// TIA Portal V20 export
VAR_GLOBAL   // PLC tag table "Servo Telgram"
   BA010AZCRDR1_UnwinderLeftAxisT_Actor_Interface_AddressIn AT %I5114.0 : "PD_TEL105_IN";
   BA010AZCRDR1_UnwinderLeftAxisT_Actor_Interface_TorqueDataAddressIn AT %I5134.0 : "PD_TEL750_IN";
   BA010AZCRDR2_UnwinderRightAxisT_Actor_Interface_AddressIn AT %I5214.0 : "PD_TEL105_IN";
   BA010AZCRDR2_UnwinderRightAxisT_Actor_Interface_TorqueDataAddressIn AT %I5234.0 : "PD_TEL750_IN";
   BA010AZCRDR3_CompensatorAxisZ_Actor_Interface_AddressIn AT %I5314.0 : "PD_TEL105_IN";
   BA010AZCRDR3_CompensatorAxisZ_Actor_Interface_TorqueDataAddressIn AT %I5344.0 : "PD_TEL750_IN";
   BA010AZCRDR4_FeedingRollAxisT_Actor_Interface_AddressIn AT %I5414.0 : "PD_TEL105_IN";
   BA010AZCRDR5_ElectordCutterAxisZ_Actor_Interface_AddressIn AT %I5514.0 : "PD_TEL105_IN";
   BA010AZCRDR6_PositionMovingAxisX_Actor_Interface_AddressIn AT %I5614.0 : "PD_TEL105_IN";
   "BA010AZCRDR7_NG&ManualInputAxisY_Actor_Interface_AddressIn" AT %I5714.0 : "PD_TEL105_IN";
   BA010AZCRDR8_MagazineAxisZ_Actor_Interface_AddressIn AT %I5814.0 : "PD_TEL105_IN";
   BA010AZCRDR9_VisionAxisZ_Actor_Interface_AddressIn AT %I5914.0 : "PD_TEL105_IN";
   BA010AZCRDR16_ReelcutRingBlow_Actor_Interface_AddressIn AT %I9906.0 : "LPD_typePDTel352In";
   BA010AZCRDR17_StackRingBlow_Actor_Interface_AddressIn AT %I9924.0 : "LPD_typePDTel352In";
   BA010AZCRDR18_StackRingBlow_Actor_Interface_AddressIn AT %I9942.0 : "LPD_typePDTel352In";
   BA010AZCRDR2_UnwinderRightAxisT_Actor_Interface_TorqueDataAddressOut AT %Q5234.0 : "PD_TEL750_OUT";
   BA010AZCRDR3_CompensatorAxisZ_Actor_Interface_TorqueDataAddressOut AT %Q5344.0 : "PD_TEL750_OUT";
   BA010AZCRDR1_UnwinderLeftAxisT_Actor_Interface_TorqueDataAddressOut AT %Q5134.0 : "PD_TEL750_OUT";
   BA010AZCRDR1_UnwinderLeftAxisT_Actor_Interface_AddressOut AT %Q5114.0 : "PD_TEL105_OUT";
   BA010AZCRDR9_VisionAxisZ_Actor_Interface_AddressOut AT %Q5914.0 : "PD_TEL105_OUT";
   BA010AZCRDR2_UnwinderRightAxisT_Actor_Interface_TAddressOut AT %Q5214.0 : "PD_TEL105_OUT";
   BA010AZCRDR8_MagazineAxisZ_Actor_Interface_AddressOut AT %Q5814.0 : "PD_TEL105_OUT";
   BA010AZCRDR3_CompensatorAxisZ_Actor_Interface_AddressOut AT %Q5314.0 : "PD_TEL105_OUT";
   BA010AZCRDR4_FeedingRollAxisT_Actor_Interface_AddressOut AT %Q5414.0 : "PD_TEL105_OUT";
   "BA010AZCRDR7_NG&ManualInputAxisY_Actor_Interface_AddressOut" AT %Q5714.0 : "PD_TEL105_OUT";
   BA010AZCRDR5_ElectordCutterAxisZ_Actor_Interface_AddressOut AT %Q5514.0 : "PD_TEL105_OUT";
   BA010AZCRDR6_PositionMovingAxisX_Actor_Interface_AddressOut AT %Q5614.0 : "PD_TEL105_OUT";
   BA010AZCRDR17_StackRingBlow_Actor_Interface_AddressOut AT %Q9924.0 : "LPD_typePDTel352Out";
   BA010AZCRDR18_StackRingBlow_Actor_Interface_AddressOut AT %Q9942.0 : "LPD_typePDTel352Out";
   BA010AZCRDR16_ReelcutRingBlow_Actor_Interface_AddressOut AT %Q9906.0 : "LPD_typePDTel352Out";
   BA010AZCRDR10_NgKickerAxisZ_Actor_Interface_AddressIn AT %I6014.0 : "PD_TEL105_IN";
   BA010AZCRDR10_NgKickerAxisZ_Actor_Interface_AddressOut AT %Q6014.0 : "PD_TEL105_OUT";
   BA010AZCRDR10_NgKickerAxisZ_Actor_Interface_TorqueDataAddressIn AT %I476.0 : "PD_TEL750_IN";
   BA010AZCRDR10_NgKickerAxisZ_Actor_Interface_TorqueDataAddressOut AT %Q476.0 : "PD_TEL750_OUT";
   BA010AZCRDR11_PassKickerAxisZ_Actor_Interface_AddressIn AT %I6114.0 : "PD_TEL105_IN";
   BA010AZCRDR11_PassKickerAxisZ_Actor_Interface_AddressOut AT %Q6114.0 : "PD_TEL105_OUT";
   BA010AZCRDR11_PassKickerAxisZ_Actor_Interface_TorqueDataAddressIn AT %I702.0 : "PD_TEL750_IN";
   BA010AZCRDR11_PassKickerAxisZ_Actor_Interface_TorqueDataAddressOut AT %Q702.0 : "PD_TEL750_OUT";
   BA010AZCRDR12_CutConveyorAxisB_Actor_Interface_AddressIn AT %I6214.0 : "PD_TEL105_IN";
   BA010AZCRDR12_CutConveyorAxisB_Actor_Interface_AddressOut AT %Q6214.0 : "PD_TEL105_OUT";
   BA010AZCRDR12_CutConveyorAxisB_Actor_Interface_TorqueDataAddressIn AT %I6234.0 : "PD_TEL750_IN";
   BA010AZCRDR12_CutConveyorAxisB_Actor_Interface_TorqueDataAddressOut AT %Q6234.0 : "PD_TEL750_OUT";
   BA010AZCRDR13_NgConveyorAxisB_Actor_Interface_AddressIn AT %I6314.0 : "PD_TEL105_IN";
   BA010AZCRDR13_NgConveyorAxisB_Actor_Interface_AddressOut AT %Q6314.0 : "PD_TEL105_OUT";
   BA010AZCRDR13_NgConveyorAxisB_Actor_Interface_TorqueDataAddressIn AT %I6334.0 : "PD_TEL750_IN";
   BA010AZCRDR13_NgConveyorAxisB_Actor_Interface_TorqueDataAddressOut AT %Q6334.0 : "PD_TEL750_OUT";
   BA010AZCRDR14_Stack1ConveyorAxisB_Actor_Interface_AddressIn AT %I6414.0 : "PD_TEL105_IN";
   BA010AZCRDR14_Stack1ConveyorAxisB_Actor_Interface_AddressOut AT %Q6414.0 : "PD_TEL105_OUT";
   BA010AZCRDR14_Stack1ConveyorAxisB_Actor_Interface_TorqueDataAddressIn AT %I6434.0 : "PD_TEL750_IN";
   BA010AZCRDR14_Stack1ConveyorAxisB_Actor_Interface_TorqueDataAddressOut AT %Q6434.0 : "PD_TEL750_OUT";
   BA010AZCRDR15_Stack2ConveyorAxisB_Actor_Interface_AddressIn AT %I6514.0 : "PD_TEL105_IN";
   BA010AZCRDR15_Stack2ConveyorAxisB_Actor_Interface_AddressOut AT %Q6514.0 : "PD_TEL105_OUT";
   BA010AZCRDR15_Stack2ConveyorAxisB_Actor_Interface_TorqueDataAddressIn AT %I6534.0 : "PD_TEL750_IN";
   BA010AZCRDR15_Stack2ConveyorAxisB_Actor_Interface_TorqueDataAddressOut AT %Q6534.0 : "PD_TEL750_OUT";
END_VAR
